FUNCTION F_Concat4 : STRING(255)
VAR_INPUT
	String1 : STRING(255);
	String2 : STRING(255);
	String3 : STRING(255);
	String4 : STRING(255);
END_VAR
VAR
END_VAR

F_Concat4 := F_CONCAT3(String2,String3,String4);
F_Concat4 := CONCAT(String1,F_Concat4);

END_FUNCTION

(* stored: Version 1.1.0.1, ProductVersion 3.1.4022.16
   POU F_Concat4: Id {4ba0ae21-62c3-4e90-a1f2-1b2dda1115c2}, SpecialFunc None *)
